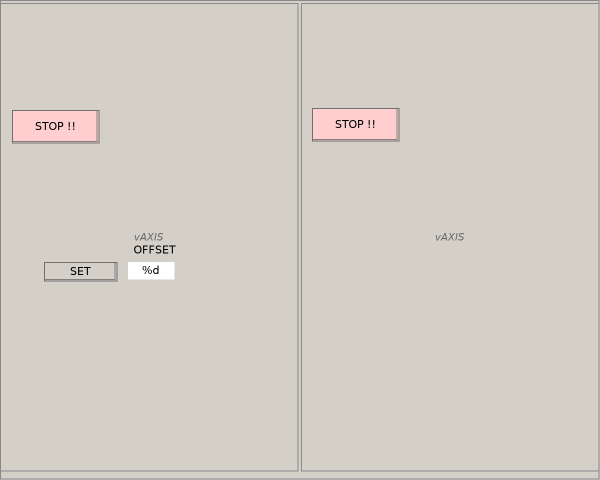
VISUALIZATION vAXES1  // 600x480
    Frame (0,3 298x468)
        shows vAXIS(vAxis := LIFT1)
    Frame (301,3 298x468)
        shows vAXIS(vAxis := XY1)
    Textfield (127,261 48x19), "%d", text variable: iOFFSET1
        OnMouseDown: write the text variable via Default
    Label (125,239 59x22), "OFFSET"
    Button (12,110 87x33), "STOP !!"
        OnMouseDown: execute { ACTION1.bSTOP_ALL:=TRUE; }
    Button (312,108 87x33), "STOP !!"
        OnMouseDown: execute { ACTION1.bSTOP_ALL:=TRUE; }
    Button (44,262 73x19), "SET"
        tap bWP_Start
END_VISUALIZATION

(* stored: Version 1.1.0.1, ProductVersion 3.1.4024.12
   Visu vAXES1: Id {6479e6f4-51f7-4978-a997-a1a308768062} *)
